{attribute 'qualified_only'}
{attribute 'strict'}
TYPE E_TestFunctionBlockRunState :
(
    IDLE := 0,
	RUNNING := 1,
    FINISHED := 2
) USINT;
END_TYPE

(* stored: Version 1.1.0.1, ProductVersion 3.1.4022.12
   DUT E_TestFunctionBlockRunState: Id {d610d037-ee39-449d-9dc9-2e1f8303e75d} *)
